{attribute 'GeneratedUsingTerminal: EJ7211-0011-0026'}
{attribute addProperty BoxType "EJ7211-0011-0026"}
{attribute addProperty Id "Target_velocityAT %Q*DINT4"}
{attribute addProperty CRC "145315899"}
{attribute addProperty Size "4"}
TYPE DS402_Target_velocity_08A9583B :
STRUCT
	{attribute addProperty Name "Target_velocity"}
	Target_velocity AT %Q* : DINT;
END_STRUCT
END_TYPE

(* stored: Version 1.2.0.0, ProductVersion 3.1.4024.9
   DUT DS402_Target_velocity_08A9583B: Id {b4a4d981-d960-4133-965c-86b7adc2e705} *)
